FUNCTION_BLOCK List_TestSuite EXTENDS TcUnit.FB_TestSuite
VAR
END_VAR

CheckAddAt();
CheckAddFirst();
CheckAddItem();
CheckAddLast();
CheckClear();
CheckContains();
CheckCopyTo();
CheckCopyToLocation();
CheckCount();
CheckGetByIndexInBounds();
CheckGetByIndexNoItems();
CheckGetByIndexOutOfBounds();
CheckImplementsICollection();
CheckImplementsIList();
CheckRemoveAtInBounds();
CheckRemoveAtNoItems();
CheckRemoveAtOutOfBounds();
CheckRemoveFirstShiftUp();
CheckRemoveNonExisting();
CheckRemoveSecondShiftUp();
CheckReturnsEnumerator();
CheckTryGetIndexOfExistingItem();
CheckTryGetIndexOfNonExistingItem();

METHOD PRIVATE CheckAddAt
VAR
	in1 : INT := 123;
	in2 : INT := 456;
	in3 : INT := 789;
	out : INT;
	result : BOOL;
	expected : INT := 789;
	list : List(4);
END_VAR
TEST('ListTests_CheckAddAt');

list.AddFirst(in1);
list.AddFirst(in2);

list.AddAt(1, in3);
list.GetByIndex(1, out);

AssertEquals(expected, out, 'Did not produce the expected result');

TEST_FINISHED();
END_METHOD

METHOD PRIVATE CheckAddFirst
VAR
	in1 : INT := 123;
	in2 : INT := 456;
	in3 : INT := 789;
	out : INT;
	result : BOOL;
	expected : INT := 789;
	list : List(4);
END_VAR
TEST('ListTests_CheckAddFirst');

list.AddLast(in1);
list.AddLast(in2);

list.AddFirst(in3);
result := list.GetByIndex(0, out);

AssertTrue(result, 'GetByIndex returned false');

AssertEquals(expected, out, 'Did not produce the expected result');

TEST_FINISHED();
END_METHOD

METHOD PRIVATE CheckAddItem
VAR
	in1 : INT := 123;
	in2 : INT := 456;
	in3 : INT := 789;
	out : INT;
	expected : INT := 789;
	list : List(4);
END_VAR
TEST('ListTests_CheckAddItem');

list.AddItem(in1);
list.AddItem(in2);
list.AddItem(in3);

list.GetByIndex(2, out);

AssertEquals(expected, out, 'Did not produce the expected result');

TEST_FINISHED();
END_METHOD

METHOD PRIVATE CheckAddLast
VAR
	in1 : INT := 123;
	in2 : INT := 456;
	in3 : INT := 789;
	out : INT;
	result : BOOL;
	expected : INT := 789;
	list : List(4);
END_VAR
TEST('ListTests_CheckAddLast');

list.AddFirst(in1);
list.AddFirst(in2);

list.AddLast(in3);
result := list.GetByIndex(2, out);

AssertTrue(result, 'GetByIndex returned false');

AssertEquals(expected, out, 'Did not produce the expected result');

TEST_FINISHED();
END_METHOD

METHOD PRIVATE CheckClear
VAR
	in1 : INT := 123;
	in2 : INT := 456;
	in3 : INT := 789;
	expected : INT := 789;
	out : INT;
	list : List(4);
END_VAR
TEST('ListTests_CheckClear');

list.AddItem(in1);
list.AddItem(in2);

list.Clear();
list.AddItem(in3);

list.GetByIndex(0, out);

AssertEquals(expected, out, 'Did not produce the expected result');

TEST_FINISHED();
END_METHOD

METHOD PRIVATE CheckContains
VAR
	in1 : INT := 123;
	in2 : INT := 456;
	in3 : INT := 789;
	result : BOOL;
	list : List(4);
END_VAR
TEST('ListTests_CheckContains');

list.AddItem(in1);
list.AddItem(in2);
list.AddItem(in3);

result := list.Contains(in2);

AssertTrue(result, 'Contains returned false while item should be in collection');

TEST_FINISHED();
END_METHOD

METHOD PRIVATE CheckCopyTo
VAR
	in1 : INT := 123;
	in2 : INT := 456;
	in3 : INT := 789;
	out : ARRAY [0..2] OF INT;
	expected : ARRAY [0..2] OF INT := [789,456,123];
	list : List(4);
END_VAR
TEST('ListTests_CheckCopyTo');

// @TEST-FIXTURE
list.AddFirst(in1); // (first->) 123 (<-last)
list.AddFirst(in2); // (first->) 456, 123 (<-last)
list.AddFirst(in3); // (first->) 789, 456, 123 (<-last)

// @TEST-RUN
list.CopyTo(out);

// @TEST-ASSSERT
AssertEquals(
	Expected := expected,
	Actual := out,
	Message := 'Did not produce the expected result'
);

TEST_FINISHED();
END_METHOD

METHOD PRIVATE CheckCopyToLocation
VAR
	in1 : INT := 123;
	in2 : INT := 456;
	in3 : INT := 789;
	out : ARRAY [0..2] OF INT;
	expected : ARRAY [0..2] OF INT := [789,456,123];
	list : List(4);
END_VAR
TEST('ListTests_CheckCopyToLocation');

// @TEST-FIXTURE
list.AddFirst(in1); // (first->) 123 (<-last)
list.AddFirst(in2); // (first->) 456, 123 (<-last)
list.AddFirst(in3); // (first->) 789, 456, 123 (<-last)

// @TEST-RUN
list.CopyToLocation(ADR(out),SIZEOF(out));

// @TEST-ASSSERT
AssertEquals(
	Expected := expected,
	Actual := out,
	Message := 'Did not produce the expected result'
);

TEST_FINISHED();
END_METHOD

METHOD PRIVATE CheckCount
VAR
	in1 : INT := 123;
	in2 : INT := 456;
	in3 : INT := 789;
	expected : ULINT := 3;
	out : ULINT;
	list : List(4);
END_VAR
TEST('ListTests_CheckCount');

list.AddItem(in1);
list.AddItem(in2);
list.AddItem(in3);

out := list.Count;

AssertEquals(expected, out, 'Did not prodocue the expected result');

TEST_FINISHED();
END_METHOD

METHOD PRIVATE CheckGetByIndexInBounds
VAR
	in1 : INT := 123;
	in2 : INT := 456;
	in3 : INT := 789;
	out : INT;
	result : BOOL;
	list : List(4);
END_VAR
TEST('ListTests_CheckGetByIndexInBounds_ReturnsTrue');

list.AddItem(in1); //Index 0
list.AddItem(in2); //Index 1
list.AddItem(in3); //Index 2

result := list.GetByIndex(1, out);

AssertTRUE(result, 'GetByIndex returned FALSE while the index is populated');

AssertEquals(in2, out, 'GetByIndex retrieved different value than expected');

TEST_FINISHED();
END_METHOD

METHOD PRIVATE CheckGetByIndexNoItems
VAR
	out : INT;
	result : BOOL;
	list : List(4);
END_VAR
TEST('ListTests_CheckGetByIndexNoItems_ReturnsFalse');

result := list.GetByIndex(0, out);

AssertFalse(result, 'GetByIndex returned TRUE while no items exist');

TEST_FINISHED();
END_METHOD

METHOD PRIVATE CheckGetByIndexOutOfBounds
VAR
	in1 : INT := 123;
	in2 : INT := 456;
	in3 : INT := 789;
	out : INT;
	result : BOOL;
	list : List(4);
END_VAR
TEST('ListTests_CheckGetByIndexOutOfBounds_ReturnsFalse');

list.AddItem(in1); //Index 0
list.AddItem(in2); //Index 1
list.AddItem(in3); //Index 2

result := list.GetByIndex(3, out);

AssertFalse(result, 'GetByIndex returned TRUE while the index is not populated');

TEST_FINISHED();
END_METHOD

METHOD PRIVATE CheckImplementsICollection
VAR
	list : List(4);
    collection : I_Collection := list;
    result : BOOL;
END_VAR
TEST('ListTests_CheckImplementsICollection');

result := collection <> 0;

AssertTrue(result, 'Did not implement ICollection');

TEST_FINISHED();
END_METHOD

METHOD PRIVATE CheckImplementsIList
VAR
	list : List(4);
    iList : I_List := list;
    result : BOOL;
END_VAR
TEST('ListTests_CheckImplementsIList');

// @TEST-FIXTURE

// @TEST-RUN
result := iList <> 0;

// @TEST-ASSSERT
AssertTrue(Condition := result,
    Message := 'Did not implement IList');

TEST_FINISHED();
END_METHOD

METHOD PRIVATE CheckRemoveAtInBounds
VAR
	in1 : INT := 123;
	in2 : INT := 456;
	in3 : INT := 789;
	out : INT;
	result : BOOL;
	list : List(4);
END_VAR
TEST('ListTests_CheckRemoveAtInBounds_ShouldRemoveAndShiftUp');

list.AddItem(in1); //Index 0
list.AddItem(in2); //Index 1
list.AddItem(in3); //Index 2

list.RemoveAt(0);

result := list.GetByIndex(0, out);

AssertTrue(result, 'Couldnt get first item');

AssertEquals(in2, out, 'Array didnt shift up items');

TEST_FINISHED();
END_METHOD

METHOD PRIVATE CheckRemoveAtNoItems
VAR
	out : INT;
	result : BOOL;
	list : List(4);
END_VAR
TEST('ListTests_CheckRemoveAtNoItems_ReturnsFalse');

result := list.RemoveAt(0);

AssertFalse(result, 'RemoveAt returned true while there was nothing to remove');

TEST_FINISHED();
END_METHOD

METHOD PRIVATE CheckRemoveAtOutOfBounds
VAR
	in1 : INT := 123;
	in2 : INT := 456;
	in3 : INT := 789;
	out : INT;
	result : BOOL;
	list : List(4);
END_VAR
TEST('ListTests_CheckRemoveAtOutOfBounds_ReturnsFalse');

list.AddItem(in1); //Index 0
list.AddItem(in2); //Index 1
list.AddItem(in3); //Index 2

result := list.RemoveAt(3);

AssertFalse(result, 'RemoveAt returned true while remove was out of bounds');

TEST_FINISHED();
END_METHOD

METHOD PRIVATE CheckRemoveFirstShiftUp
VAR
	in1 : INT := 123;
	in2 : INT := 456;
	in3 : INT := 789;
	out : INT;
	result : BOOL;
	list : List(4);
END_VAR
TEST('ListTests_CheckRemoveFirst_ShiftUp');

list.AddItem(in1); //Index 0
list.AddItem(in2); //Index 1
list.AddItem(in3); //Index 2

list.RemoveItem(in1);

result := list.GetByIndex(0, out);

AssertTrue(result, 'Coulndt get first item');

AssertEquals(in2, out, 'Array didnt shift up items');

TEST_FINISHED();
END_METHOD

METHOD PRIVATE CheckRemoveNonExisting
VAR
	in1 : INT := 123;
	in2 : INT := 456;
	in3 : INT := 789;
	out : INT;
	result : BOOL;
	list : List(4);
END_VAR
TEST('ListTests_CheckRemoveNonExisting_ReturnsFalse');

list.AddItem(in1); //Index 0
list.AddItem(in2); //Index 1

result := list.RemoveItem(in3);

AssertFalse(result, 'GetByIndex returned something');

TEST_FINISHED();
END_METHOD

METHOD PRIVATE CheckRemoveSecondShiftUp
VAR
	in1 : INT := 123;
	in2 : INT := 456;
	in3 : INT := 789;
	out : INT;
	result : BOOL;
	list : List(4);
END_VAR
TEST('ListTests_CheckRemoveSecond_ShiftUp');

list.AddItem(in1); //Index 0
list.AddItem(in2); //Index 1
list.AddItem(in3); //Index 2

list.RemoveItem(in2);

result := list.GetByIndex(1, out);

AssertTrue(result, 'Coulndt get first item');

AssertEquals(in3, out, 'Array didnt shift up items');

TEST_FINISHED();
END_METHOD

METHOD PRIVATE CheckReturnsEnumerator
VAR
	in1 : INT := 123;
	in2 : INT := 456;
	in3 : INT := 789;
	list : List(4);
	enumerator : I_ForwardEnumerator;
	enumerable : I_Enumerable := list;
	result : BOOL;
END_VAR
TEST('ListTests_CheckLinkedListReturnsEnumerator');

// @TEST-FIXTURE
list.AddItem(in1); // (first->) 123 (<-last)
list.AddItem(in2); // (first->) 456, 123 (<-last)
list.AddItem(in3); // (first->) 789, 456, 123 (<-last)

// @TEST-RUN
result := enumerable <> 0;

enumerator := list.GetEnumerator();

// @TEST-ASSSERT
AssertTrue(result, 'Did not implement IEnumerable');

AssertTrue(
	Condition := (enumerator <> 0),
	Message := 'Did not return an enumerator'
);

// @TEST-DISPOSE
enumerator.Dispose();

TEST_FINISHED();
END_METHOD

METHOD PRIVATE CheckTryGetIndexOfExistingItem
VAR
	in1 : INT := 123;
	in2 : INT := 456;
	in3 : INT := 789;
	out : UDINT;
	expected : UDINT := 1;
	result : BOOL;
	list : List(4);
END_VAR
TEST('ListTests_CheckTryGetIndexOfExistingItem_ReturnsIndex');

list.AddItem(in1); //Index 0
list.AddItem(in2); //Index 1
list.AddItem(in3); //Index 2

result := list.TryGetIndexOf(in2, index => out);

AssertTrue(result, 'TryGetIndexOf returned false on a existing item');

AssertEquals(out, expected, 'The index is not the expected index');

TEST_FINISHED();
END_METHOD

METHOD PRIVATE CheckTryGetIndexOfNonExistingItem
VAR
	in1 : INT := 123;
	in2 : INT := 456;
	in3 : INT := 789;
	out : UDINT;
	result : BOOL;
	list : List(4);
END_VAR
TEST('ListTests_CheckTryGetIndexOfNonExistingItem_ReturnsIndex');

list.AddItem(in1); //Index 0
list.AddItem(in2); //Index 1

result := list.TryGetIndexOf(in3, index => out);

AssertFalse(result, 'TryGetIndexOf returned true on a non-existing item');

TEST_FINISHED();
END_METHOD

END_FUNCTION_BLOCK

(* stored: Version 1.1.0.1, ProductVersion 3.1.4024.12
   POU List_TestSuite: Id {687abae4-6464-4e6f-b6bc-2179a67dd6ef}, SpecialFunc None
   Method CheckAddAt: Id {4199ef1e-4f5e-43c7-ba81-fe66d0a50263}
   Method CheckAddFirst: Id {dc616732-ccec-4a50-a24e-6046ca902467}
   Method CheckAddItem: Id {53909bfa-2a23-432c-b757-416cc9a28880}
   Method CheckAddLast: Id {d8ce7920-f4a3-4ee7-bfb0-5ec4529b25fe}
   Method CheckClear: Id {7bdd9076-8eb2-4cff-91b2-e91622dce2a8}
   Method CheckContains: Id {41106fd9-1ecf-4862-9978-93774600dc73}
   Method CheckCopyTo: Id {b0184d3d-3b2e-4473-a2b5-bcd866b47371}
   Method CheckCopyToLocation: Id {3e2ea42d-a96e-4b82-9432-3dccf597c7b7}
   Method CheckCount: Id {e7d8659d-642d-4fc5-bd70-73d1275abde8}
   Method CheckGetByIndexInBounds: Id {ed595b19-d81c-4103-b5b9-317253636f87}
   Method CheckGetByIndexNoItems: Id {b54c7e02-1794-445e-93a2-5e10dd961aa3}
   Method CheckGetByIndexOutOfBounds: Id {a1f9bb81-24dc-40fb-9530-878e73a45762}
   Method CheckImplementsICollection: Id {a6d761ea-1ba3-4a5f-b0c7-b9c1be384a89}
   Method CheckImplementsIList: Id {ab3222f8-29e7-4132-b4e8-8f60d299cce9}
   Method CheckRemoveAtInBounds: Id {71fd981e-ebf6-4028-81ff-00b5119c6397}
   Method CheckRemoveAtNoItems: Id {5eb1d086-e5fd-43f5-a685-8086d855e5ed}
   Method CheckRemoveAtOutOfBounds: Id {14964f08-9d5c-4b83-9628-56623c1f3cc1}
   Method CheckRemoveFirstShiftUp: Id {a265e32b-e122-4925-81d7-d57bfffbd7a3}
   Method CheckRemoveNonExisting: Id {f71d7acd-ac3b-434f-88a3-9c9fa917f6bb}
   Method CheckRemoveSecondShiftUp: Id {a9c35f26-ec4f-480d-81e6-f13903eac4e4}
   Method CheckReturnsEnumerator: Id {d40571a0-acd3-4f34-a952-5924360dee95}
   Method CheckTryGetIndexOfExistingItem: Id {bd87f2e8-54dc-42d5-8914-6d113f39282d}
   Method CheckTryGetIndexOfNonExistingItem: Id {43467fde-fa83-4538-a1b8-7f87bcaf7d56} *)
